{attribute 'linkalways'} 
{attribute 'no_explicit_call' := 'This FB is a CLASS and must be accessed using methods or properties'}
{attribute 'enable_dynamic_creation'}
FUNCTION_BLOCK _ETcVnCalibrationPatternOrigin EXTENDS EnumDatatypeBase
VAR
	localData : ETcVnCalibrationPatternOrigin;
	activeData : REFERENCE TO ETcVnCalibrationPatternOrigin;
	enumBaseDatatype : _DINT(localData);
END_VAR

METHOD PRIVATE AddLocalEnumeration
VAR_INPUT
	Enumeration : T_MAXSTRING;
	Value : ETcVnCalibrationPatternOrigin;
END_VAR
AddEnumeration(Enumeration, Value);
END_METHOD

PROPERTY PUBLIC Address : PVOID
GET
Address := ADR(activeData);
END_GET
END_PROPERTY

METHOD PUBLIC ClearReference
VAR_INPUT
END_VAR
activeData REF= localData;
SetBaseDatatypeReference();
END_METHOD

METHOD PUBLIC Clone : I_Datatype
VAR
    pClone : POINTER TO _ETcVnCalibrationPatternOrigin;
END_VAR
pClone := __NEW(_ETcVnCalibrationPatternOrigin(InitialValue := Value));
Clone := pClone^;
END_METHOD

METHOD FB_init : BOOL
VAR_INPUT
	bInitRetains : BOOL; // if TRUE, the retain variables are initialized (warm start / cold start)
	bInCopyCode : BOOL;  // if TRUE, the instance afterwards gets moved into the copy code (online change)
	InitialValue : ETcVnCalibrationPatternOrigin;
END_VAR
localData := InitialValue;
AddBaseDatatype(enumBaseDatatype);
ClearReference();

AddLocalEnumeration('TCVN_CPO_TOPLEFT', ETcVnCalibrationPatternOrigin.TCVN_CPO_TOPLEFT);
AddLocalEnumeration('TCVN_CPO_TOPCENTER', ETcVnCalibrationPatternOrigin.TCVN_CPO_TOPCENTER);
AddLocalEnumeration('TCVN_CPO_TOPRIGHT', ETcVnCalibrationPatternOrigin.TCVN_CPO_TOPRIGHT);
AddLocalEnumeration('TCVN_CPO_CENTERLEFT', ETcVnCalibrationPatternOrigin.TCVN_CPO_CENTERLEFT);
AddLocalEnumeration('TCVN_CPO_CENTER', ETcVnCalibrationPatternOrigin.TCVN_CPO_CENTER);
AddLocalEnumeration('TCVN_CPO_CENTERRIGHT', ETcVnCalibrationPatternOrigin.TCVN_CPO_CENTERRIGHT);
AddLocalEnumeration('TCVN_CPO_BOTTOMLEFT', ETcVnCalibrationPatternOrigin.TCVN_CPO_BOTTOMLEFT);
AddLocalEnumeration('TCVN_CPO_BOTTOMCENTER', ETcVnCalibrationPatternOrigin.TCVN_CPO_BOTTOMCENTER);
AddLocalEnumeration('TCVN_CPO_BOTTOMRIGHT', ETcVnCalibrationPatternOrigin.TCVN_CPO_BOTTOMRIGHT);
END_METHOD

PROPERTY PUBLIC Identifier : T_MAXSTRING
GET
Identifier := 'ETcVnCalibrationPatternOrigin';
END_GET
END_PROPERTY

METHOD IsEnumeratorValueEqual : BOOL
VAR_INPUT
	Enumerator : I_KeyValueForwardEnumerator;
END_VAR
VAR
	storedValue : ETcVnCalibrationPatternOrigin;
END_VAR
IF NOT Enumerator.TryGet(storedValue) THEN
	RETURN;
END_IF

IsEnumeratorValueEqual := storedValue = activeData;
END_METHOD

METHOD PUBLIC MakeReferenceTo
VAR_INPUT
	ReferenceTarget : REFERENCE TO ETcVnCalibrationPatternOrigin;
END_VAR
activeData REF= ReferenceTarget;
SetBaseDatatypeReference();
END_METHOD

METHOD PROTECTED SetBaseDatatypeReference
VAR_INPUT
END_VAR
enumBaseDatatype.MakeReferenceTo(activeData);
END_METHOD

PROPERTY PUBLIC Size : UDINT
GET
Size := SIZEOF(activeData);
END_GET
END_PROPERTY

METHOD TryMakeReferenceTo : BOOL
VAR_INPUT
	Target : I_Datatype;
END_VAR
VAR
	pTargetData : POINTER TO ETcVnCalibrationPatternOrigin;
END_VAR
IF NOT IsEquivalentTo(Target) THEN
	RETURN;
END_IF

pTargetData := Target.Address;
activeData REF= pTargetData^;
SetBaseDatatypeReference();
TryMakeReferenceTo := TRUE;
END_METHOD

PROPERTY PUBLIC Value : ETcVnCalibrationPatternOrigin
GET
Value := activeData;
END_GET
SET
activeData := Value;
END_SET
END_PROPERTY

END_FUNCTION_BLOCK

(* stored: Version 1.1.0.1, ProductVersion 3.1.4024.13
   POU _ETcVnCalibrationPatternOrigin: Id {4ccacb9b-3608-4251-91bc-8ded518735ef}, SpecialFunc None
   Folder Core: Id {6375380d-eff3-08e0-081a-65c9995b39a4}
   Folder Protected: Id {8110a88e-9c27-0937-17a4-74c764766314}
   Folder Customize: Id {bc2750f5-0c51-0590-2090-840b30e811ad}
   Folder Constructor: Id {e529e4a4-f9fc-4a9d-93cc-d6bcb568dcb5}
   Folder Private: Id {bb9d4f1c-eae1-44ee-9f00-e642cebfc9c9}
   Folder Protected: Id {2b0221f8-dd26-44c0-8a83-9b22d28fbe8e}
   Method AddLocalEnumeration: Id {ed8ab352-0b5f-4483-adfa-08e25f8e6c31}
   Property Address: Id {4f399cb7-da09-0570-2971-5fcd26f80176}
   Get Get: Id {d8927b6f-cc1c-07f9-2388-43a1575e42a4}
   Method ClearReference: Id {c39d3680-5fcf-0855-2bd0-e0c26440aedf}
   Method Clone: Id {63f8ca8d-fa44-4943-98c5-8b114c6b8a89}
   Method FB_init: Id {f160c241-eedd-4716-a78f-436960b8b1ba}
   Property Identifier: Id {43f86303-8cae-4e11-bda1-191751e29d86}
   Get Get: Id {aef3b22d-718f-4c89-a278-aa45d9950d93}
   Method IsEnumeratorValueEqual: Id {fcaec953-932c-45b1-a554-94bb948fbb98}
   Method MakeReferenceTo: Id {86540879-d2ed-4e31-b1fa-19c67851f2c1}
   Method SetBaseDatatypeReference: Id {2892c9d3-66b5-0c47-1be8-5d4f885fb318}
   Property Size: Id {4f4e3d57-4dc3-0a37-0b69-1f83dd97b439}
   Get Get: Id {f021ca6a-a829-01ed-0326-ada300723ce8}
   Method TryMakeReferenceTo: Id {53ddb35a-a29b-46ea-8c77-992581344705}
   Property Value: Id {00c9fdaa-0053-431b-b86c-08ed8ffafbd3}
   Get Get: Id {b4f3de94-7591-4140-92d4-24ddcf9fca0c}
   Set Set: Id {1acd0613-d8cb-4181-8c66-2a716c694462} *)
